(* IEC 61131-3 sources: plcassist-cli/packages/volt-lsp-iec/test-corpus/pro2193/Device/Plc Logic/Application/03 Hardware Units/31 SER/31.30 - Z Units/Base, 3 files *)

(* ---- IZUnit_Stacking_Commands.itf ---- *)
// Commands specific for an Z Unit
INTERFACE IZUnit_Stacking_Commands

// Await stacking delay
METHOD PUBLIC AwaitDelay : BOOL
VAR_INPUT
	firstStack	: BOOL;
END_VAR
END_METHOD

// Move down to place products on the stack
METHOD PUBLIC MoveDown : BOOL
VAR_INPUT
	stackIndex			: UINT;	// Actual number on the stack (stackingheight)
END_VAR
END_METHOD

// Start to move down. Wait above the stack if the conveyor is not ready.
METHOD PUBLIC MoveDown_Start : BOOL
VAR_INPUT
	highestStackIndex		: UINT;	// Stackingheight of a complete stack (to rotate above)
END_VAR
END_METHOD

// Move up to final position
METHOD PUBLIC MoveUp : BOOL
END_METHOD

// Start to move up from the stack
METHOD PUBLIC MoveUp_Start : BOOL
VAR_INPUT
	stackIndex			: UINT;	// Stackingheight to rotate above. Can be either act stackheight, or max stackheight
END_VAR
END_METHOD

// Returns the products that are currently stacked by the Z Unit
METHOD PUBLIC ProductData_Get : ProductType
VAR_INPUT
	product			: UINT;
	clearData		: BOOL := FALSE;	// Optional: Clear data of the product that is being transferred.
END_VAR
END_METHOD

// Product transfer is complete, ready for stacking (or something else)
{attribute 'monitoring':='call'}
PROPERTY ReadyForStacking : BOOL;
GET
END_GET
END_PROPERTY

END_INTERFACE

(* ---- IZUnit_Transfer_Commands.itf ---- *)
// Commands specific for an Z Unit
INTERFACE IZUnit_Transfer_Commands
EXTENDS IModuleTransferComplete, IModuleManualControlEnabled

// Receive a product status
METHOD PUBLIC CopyProductStatus : BOOL
VAR_INPUT
	takeoverPos		: INT;
	productNo		: INT(1..TO_INT(GVL_Constants.ChainProductsForZUnit));
	product			: ProductType;
END_VAR
END_METHOD

// Receive a certain amount of products by vacuum or clamps. Parameter indicates which product is received. Returns index of products that are actually transferred.
METHOD PUBLIC GetProducts : BOOL
VAR_INPUT
	vacuumIndex		: REFERENCE TO WORD;	// 0: All vacuums, bit 1: Vacuum 1, bit 2: Vacuum 2, etc.
END_VAR
END_METHOD

// Move to a certain Takeover position
METHOD PUBLIC MoveToTakeover : BOOL
VAR_INPUT
	takeoverPosition		: INT;	// 0: invalid, 1: Takeover pos 1, etc.
END_VAR
END_METHOD

// Z unit is ready to receive products
{attribute 'monitoring':='call'}
PROPERTY ReadyForTransfer : BOOL;
GET
END_GET
END_PROPERTY

END_INTERFACE

(* ---- ZUnit_BaseFB.fb ---- *)
{attribute 'symbol' := 'none'}
FUNCTION_BLOCK ABSTRACT ZUnit_BaseFB
EXTENDS ModuleWithBrakedServoBaseFB
VAR_IN_OUT
	Data						: ZUnit_Base_Data;
END_VAR
VAR//VISU
	{attribute 'symbol' := 'read'}	rMaxTorqueMovingUp			: REAL;			// Max torque while moving up (in Nm)
END_VAR
VAR
	ReadMachineData				: L_MC1P.L_MC1P_ReadMachineData;

	// Private backing fields for properties
	{attribute 'hide'}	_readyForStacking			: BOOL;
	{attribute 'hide'}	_readyForTransfer			: BOOL;
END_VAR
VAR CONSTANT
	NumberOfTakeoverPositions	: USINT	:= ZUnits.NumberOfTakeoverPositions;
END_VAR

SUPER^(
	AxisRef				:= AxisRef,
	DataBrink			:= DataBrink,
	coveredDistance		:= coveredDistance,
);

END_FUNCTION_BLOCK

METHOD PROTECTED Cyclic
VAR_INST
	guardPosition				: ARRAY[1..4] OF GuardRealFB(									moduleHandler	:= ModuleHandler);
	attachPosition				: ARRAY[1..1] OF AttachPosToButtonFB(							drive			:= Drive);
	guardTakeoverPosition		: ARRAY[1..NumberOfTakeoverPositions] OF GuardRealFB(			moduleHandler	:= ModuleHandler);
	attachTakeoverPosition		: ARRAY[1..NumberOfTakeoverPositions] OF AttachPosToButtonFB(	drive			:= Drive);
END_VAR
VAR
	i							: USINT;
END_VAR
ReadMachineData(
	Axis					:= AxisRef,
	xEnable					:= TRUE,
	xValid					=> ,
	xBusy					=> ,
	xError					=> ,
	eErrorID				=> ,
	lrFeedconstant			=> ,
	dwGearDenominator		=> ,
	dwGearNumerator			=> ,
	dwAddGearDenominator	=> ,
	dwAddGearNumerator		=> ,
	dwPosResolution			=> ,
	xOrientation			=> ,
	eTraversingRange		=> ,
	lrCycleLength			=> ,
	xVirtual				=> );

// Set limits for the positions, and guard the limits
Data.FirstPart.Pos.lowerLimit						:= Arrays.Position_Largest(Data.Takeover);
Data.FirstPart.Pos.upperLimit						:= DataBrink.rSWLimitPos;

PersistentVars.RecipeVars.productPitch.lowerLimit	:= 0.1;
PersistentVars.RecipeVars.productPitch.upperLimit	:= 100;
PersistentVars.RecipeVars.productPitch.stepSize		:= 0.1;

PersistentVars.RecipeVars.productHeight.lowerLimit	:= 1;
PersistentVars.RecipeVars.productHeight.upperLimit	:= 500;
PersistentVars.RecipeVars.productHeight.stepSize	:= 2;

Data.EarlyProductReleaseDistance.lowerLimit			:= 0;
Data.EarlyProductReleaseDistance.upperLimit			:= Data.FirstPart.Pos.value - Arrays.Position_Largest(Data.Takeover);
Data.EarlyProductReleaseDistance.stepSize			:= 10;

FOR i := 1 TO NumberOfTakeoverPositions DO
	Data.Takeover[i].Pos.lowerLimit		:= DataBrink.rSWLimitNeg;
	Data.Takeover[i].Pos.upperLimit		:= Data.FirstPart.Pos.value;
	guardTakeoverPosition[i](		value := Data.Takeover[i].Pos);
	attachTakeoverPosition[i](		value := Data.Takeover[i].Pos);
END_FOR

guardPosition[1](value := Data.FirstPart.Pos);
guardPosition[2](value := PersistentVars.RecipeVars.productPitch);
guardPosition[3](value := PersistentVars.RecipeVars.productHeight);
guardPosition[4](value := Data.EarlyProductReleaseDistance);

attachPosition[1](value := Data.FirstPart.Pos);
END_METHOD

// Command to reset the module (Statemachine to zero state) in case of E-Stop
METHOD PUBLIC EStop : BOOL	// Returns true when drives are in standstill
%FOLDER Commands
ReadyForTransfer	:= FALSE;
ReadyForStacking	:= FALSE;

Drive.Quickstop(TRUE);

EStop := (Drive.Standstill OR NOT Drive.AxisEnabled) AND SUPER^.EStop();
END_METHOD

METHOD PROTECTED Initialize
SUPER^.Initialize();

DriveBrakeLogic.config.holdingTorque		:= -6;
END_METHOD

// Command to reset the module (Statemachine to zero state)
METHOD PUBLIC Stop : BOOL	// Returns true when drives are in standstill
%FOLDER Commands
IF NOT GlobalVars.Reset AND Drive.AxisEnabled AND NOT Drive.config.virtualMode THEN
	Drive.Halt();
END_IF

Stop := (Drive.Standstill OR NOT Drive.AxisEnabled) AND SUPER^.Stop();
END_METHOD

// Product transfer is complete, ready for stacking (or something else)
{attribute 'monitoring':='call'}
PROPERTY ReadyForStacking : BOOL;
%FOLDER Properties
GET
VAR
END_VAR
ReadyForStacking	:= _readyForStacking;
END_GET
SET
PROTECTED
VAR
END_VAR
_readyForStacking	:= ReadyForStacking;
END_SET
END_PROPERTY

// Z unit is ready to receive products
{attribute 'monitoring':='call'}
PROPERTY ReadyForTransfer : BOOL;
%FOLDER Properties
GET
VAR
END_VAR
ReadyForTransfer	:= _readyForTransfer;
END_GET
SET
PROTECTED
VAR
END_VAR
_readyForTransfer	:= ReadyForTransfer;
END_SET
END_PROPERTY

// Torque is mirrored when drive is mounted CW or CCW. Correct for this. Use torque for crash detection of Z Unit
{attribute 'monitoring':='call'}
PROPERTY TorqueCorrected : REAL;
%FOLDER Properties
GET
VAR
END_VAR
IF ReadMachineData.xValid AND_THEN ReadMachineData.xOrientation THEN
	TorqueCorrected	:= Drive.actTorque * -1;
ELSE
	TorqueCorrected	:= Drive.actTorque;
END_IF

// In memory of Henrie Meijer
// He always pushed to get this function in the software
END_GET
END_PROPERTY
